// Mitsubishi GX Works2 project: PartB4   PLC: FX3G

// global labels: Global1
VAR_GLOBAL
  X_10 AT X010 : BOOL;
  sen_w AT X003 : BOOL;
  sen_sp1 AT X004 : BOOL;
  sen_sm1 AT X005 : BOOL;
  Y_1 AT Y001 : BOOL;
  Y_2 AT Y002 : BOOL;
  Y_3 AT Y003 : BOOL;
  sen_t AT X006 : BOOL;
  M_0 AT Y010 : BOOL;
  TC_1 AT TC1 : BOOL;
  TS_1 AT TS1 : BOOL;
END_VAR
VAR_GLOBAL CONSTANT
  Timing1 : INT := 20;
END_VAR
VAR_GLOBAL
  TC_2 AT TC2 : BOOL;
  TS_2 AT TS2 : BOOL;
END_VAR
VAR_GLOBAL CONSTANT
  Timing2 : INT := 20;
END_VAR
VAR_GLOBAL
  sen_d3 AT X000 : BOOL;
  sen_d5 AT X001 : BOOL;
  Y_4 AT Y004 : BOOL;
END_VAR

// task Task_01 (event TRUE, interval 0, priority 31): POU_01

PROGRAM POU_01
(* structured ladder/FBD written out as ST: instructions are called as NAME(EN, inputs, outputs); _pN, _eN, _tN stand for wires *)
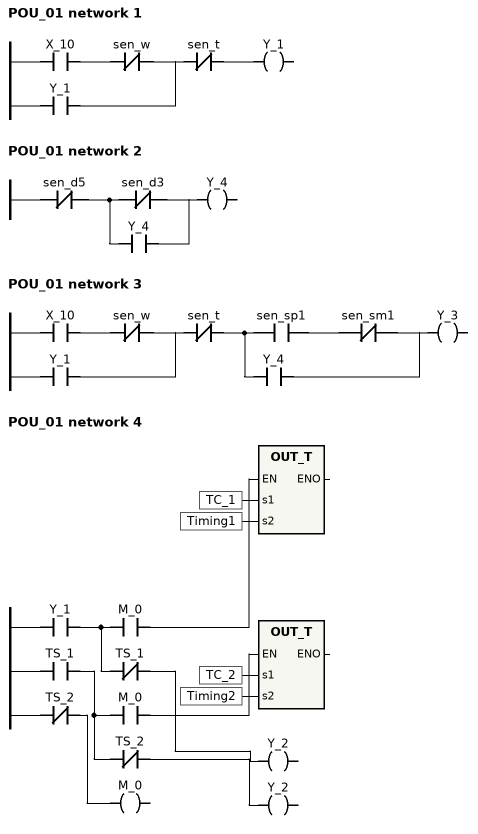
(* network 1 *)
Y_1 := ((X_10 AND NOT sen_w) OR Y_1) AND NOT sen_t;
(* network 2 *)
_p1 := NOT sen_d5;
Y_4 := (_p1 AND NOT sen_d3) OR (_p1 AND Y_4);
(* network 3 *)
_p1 := ((X_10 AND NOT sen_w) OR Y_1) AND NOT sen_t;
Y_3 := (_p1 AND sen_sp1 AND NOT sen_sm1) OR (_p1 AND Y_4);
(* network 4 *)
OUT_T(Y_1 AND M_0, TC_1, Timing1);
Y_2 := Y_1 AND NOT TS_1;
OUT_T(TS_1 AND M_0, TC_2, Timing2);
Y_2 := TS_1 AND NOT TS_2;
M_0 := NOT TS_2;
END_PROGRAM
